# EPICS substitutions: hugo/source/db/Beckhoff_3XXX/ecmcEL3174.substitutions
#Actually the scalinging is between 0..10.737V (see manual)
file "ecmc_analogInput-chX.template"
{
  pattern {CH_ID, EGU  }
          {01,    "Raw"}
          {02,    "Raw"}
          {03,    "Raw"}
          {04,    "Raw"}
}

file "ecmc_status-chX.template"
{
  pattern {CH_ID, KEY }
          {01,    "AI"}
          {02,    "AI"}
          {03,    "AI"}
          {04,    "AI"}
}
